Fanuc KAREL source: NC0029.KL

-- PROVISIONAL review KL for V940-1; original PC SHA256 8393bc4ced0f805fe74e50ed637e114a0d37e5fe415938faf5a8cfaab3dc543a
-- Incomplete behavior may be omitted. Consult companion uncertainty JSON. Do not deploy.
PROGRAM NC0029
%NOLOCKGROUP
-- UNRESOLVED_LOCAL_POOL 1 cells at code offset 3; source declarations unknown
-- DIRECT_LOCAL_WORD_ACCESS alone does not prove INTEGER, REAL, or BOOLEAN
BEGIN
  -- UNRESOLVED_PC offsets 0-8; opcodes 2B,2C,7B
  -- UNRESOLVED_PC offsets 13-20; opcodes 9D,23
  -- UNRESOLVED_PC offsets 25-42; opcodes 21,40,41,42
  -- UNRESOLVED_PC offsets 47-64; opcodes 21,40,41,42
  -- UNRESOLVED_PC offsets 69-86; opcodes 21,40,41,42
  -- UNRESOLVED_PC offsets 91-108; opcodes 21,40,41,42
  -- UNRESOLVED_PC offsets 113-130; opcodes 21,40,41,42
  -- UNRESOLVED_PC offsets 135-152; opcodes 21,40,41,42
  -- UNRESOLVED_PC offsets 157-174; opcodes 21,40,41,42
  -- UNRESOLVED_PC offsets 179-196; opcodes 21,40,41,42
  -- UNRESOLVED_PC offsets 201-218; opcodes 21,40,41,42
  -- UNRESOLVED_PC offsets 223-240; opcodes 21,40,41,42
  -- UNRESOLVED_PC offsets 245-262; opcodes 21,40,41,42
  -- UNRESOLVED_PC offsets 267-284; opcodes 21,40,41,42
  -- UNRESOLVED_PC offsets 289-306; opcodes 21,40,41,42
  -- UNRESOLVED_PC offsets 311-328; opcodes 21,40,41,42
  -- UNRESOLVED_PC offsets 333-350; opcodes 21,40,41,42
  -- UNRESOLVED_PC offsets 355-385; opcodes 21,9D,52,23,7A,40,41,42
  -- UNRESOLVED_PC offsets 390-414; opcodes 21,2E,52,23,7A,43
  -- UNRESOLVED_PC offsets 419-437; opcodes 21,2E,52,23
  -- UNRESOLVED_PC offsets 442-458; opcodes 7A,40,41,42
  -- UNRESOLVED_PC offsets 463-487; opcodes 21,2E,52,23,7A,43
  -- UNRESOLVED_PC offsets 492-510; opcodes 21,2E,52,23
  -- UNRESOLVED_PC offsets 515-531; opcodes 7A,40,41,42
  -- UNRESOLVED_PC offsets 536-560; opcodes 21,2E,52,23,7A,43
  -- UNRESOLVED_PC offsets 565-583; opcodes 21,2E,52,23
  -- UNRESOLVED_PC offsets 588-604; opcodes 7A,40,41,42
  -- UNRESOLVED_PC offsets 609-633; opcodes 21,2E,52,23,7A,43
  -- UNRESOLVED_PC offsets 638-656; opcodes 21,2E,52,23
  -- UNRESOLVED_PC offsets 661-677; opcodes 7A,40,41,42
  -- UNRESOLVED_PC offsets 682-706; opcodes 21,2E,52,23,7A,43
  -- UNRESOLVED_PC offsets 711-729; opcodes 21,2E,52,23
  -- UNRESOLVED_PC offsets 734-750; opcodes 7A,40,41,42
  -- UNRESOLVED_PC offsets 755-779; opcodes 21,2E,52,23,7A,43
  -- UNRESOLVED_PC offsets 784-802; opcodes 21,2E,52,23
  -- UNRESOLVED_PC offsets 807-823; opcodes 7A,40,41,42
  -- UNRESOLVED_PC offsets 828-852; opcodes 21,2E,52,23,7A,43
  -- UNRESOLVED_PC offsets 857-875; opcodes 21,2E,52,23
  -- UNRESOLVED_PC offsets 880-896; opcodes 7A,40,41,42
  -- UNRESOLVED_PC offsets 901-925; opcodes 21,2E,52,23,7A,43
  -- UNRESOLVED_PC offsets 930-948; opcodes 21,2E,52,23
  -- UNRESOLVED_PC offsets 953-969; opcodes 7A,40,41,42
  -- UNRESOLVED_PC offsets 974-998; opcodes 21,2E,52,23,7A,43
  -- UNRESOLVED_PC offsets 1003-1021; opcodes 21,2E,52,23
  -- UNRESOLVED_PC offsets 1026-1042; opcodes 7A,40,41,42
  -- UNRESOLVED_PC offsets 1047-1071; opcodes 21,2E,52,23,7A,43
  -- UNRESOLVED_PC offsets 1076-1094; opcodes 21,2E,52,23
  -- UNRESOLVED_PC offsets 1099-1115; opcodes 7A,40,41,42
  -- UNRESOLVED_PC offsets 1120-1144; opcodes 21,2E,52,23,7A,43
  -- UNRESOLVED_PC offsets 1149-1167; opcodes 21,2E,52,23
  -- UNRESOLVED_PC offsets 1172-1188; opcodes 7A,40,41,42
  -- UNRESOLVED_PC offsets 1193-1217; opcodes 21,2E,52,23,7A,43
  -- UNRESOLVED_PC offsets 1222-1240; opcodes 21,2E,52,23
  -- UNRESOLVED_PC offsets 1245-1261; opcodes 7A,40,41,42
  -- UNRESOLVED_PC offsets 1266-1290; opcodes 21,2E,52,23,7A,43
  -- UNRESOLVED_PC offsets 1295-1313; opcodes 21,2E,52,23
  -- UNRESOLVED_PC offsets 1318-1334; opcodes 7A,40,41,42
  -- UNRESOLVED_PC offsets 1339-1363; opcodes 21,2E,52,23,7A,43
  -- UNRESOLVED_PC offsets 1368-1386; opcodes 21,2E,52,23
  -- UNRESOLVED_PC offsets 1391-1407; opcodes 7A,40,41,42
  -- UNRESOLVED_PC offsets 1412-1436; opcodes 21,2E,52,23,7A,43
  -- UNRESOLVED_PC offsets 1441-1459; opcodes 21,2E,52,23
  -- UNRESOLVED_PC offsets 1469-1473; opcodes 7F
  -- UNRESOLVED_PC offsets 1478-1482; opcodes 27,AA
  -- UNRESOLVED_PC offsets 1487-1491; opcodes 7F
END NC0029
